INTERFACE ITF_ActuatorDecoratorTest EXTENDS ITF_Actuator

END_INTERFACE

(* stored: Version 1.1.0.1
   Itf ITF_ActuatorDecoratorTest: Id {0ef77d46-a915-0e2d-3bd0-147aa75b6a35} *)
